Fanuc KAREL source: kd00013.KL

PROGRAM KD00013
%STACKSIZE=65535
%PRIORITY=65535
%NOLOCKGROUP
VAR
I : INTEGER
J : INTEGER
B : BOOLEAN
R : REAL
S : STRING[80]
BEGIN
-- UNRESOLVED_PC line 10 opcodes [2E 9D 1A] marker_code=0
END KD00013
